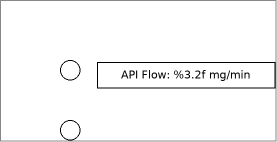
VISUALIZATION ContinuousFormulation  // 277x142
    Ellipse (60,60 20x20)
    Ellipse (60,120 20x20)
    Rectangle (97,62 178x26), "API Flow: %3.2f mg/min", text variable: IO.FT_API_PV
END_VISUALIZATION

(* stored: Version 1.1.0.1, ProductVersion 3.1.4019.2
   Visu ContinuousFormulation: Id {2716c03c-f05c-4b1d-817d-4b5595bb5f41} *)
